{attribute 'hide_all_locals'}
FUNCTION_BLOCK DisableGroup IMPLEMENTS ITask
VAR_INPUT
END_VAR
VAR_OUTPUT
END_VAR
VAR
	groupDisable			: MC_GroupDisable;
	_caGroup			: REFERENCE TO AXES_GROUP_REF;
	State: INT;
	_disableGroup : BOOL;
	_busy : BOOL;
	_error : BOOL;
	_done : BOOL;
END_VAR

CASE State OF
	0:
		IF _disableGroup THEN
			_done := FALSE;
			_error := FALSE;
			_busy := TRUE;
			groupDisable.Execute := TRUE;
			IF groupDisable.Busy THEN
				_disableGroup := FALSE;
				State := 10;
			END_IF
		END_IF
	
	10:
		IF NOT groupDisable.Busy THEN
			IF groupDisable.Done THEN
				_done := TRUE;
			ELSIF groupDisable.Error THEN
				_error := TRUE;
			END_IF
			_busy := FALSE;
			groupDisable.Execute := false;
			State := 0;
		END_IF
END_CASE


groupDisable(AxesGroup := _caGroup);

METHOD Abort : BOOL
State := 0;
groupDisable.Execute := FALSE;
Abort := true;
END_METHOD

PROPERTY Busy : BOOL
GET
Busy := _busy;
END_GET
END_PROPERTY

PROPERTY Done : BOOL
GET
Done := _done;
END_GET
END_PROPERTY

PROPERTY Error : BOOL
GET
Error := _error;
END_GET
END_PROPERTY

METHOD Execute : BOOL
Execute := _disableGroup := TRUE;
END_METHOD

METHOD FB_init : BOOL
VAR_INPUT
	bInitRetains : BOOL; // if TRUE, the retain variables are initialized (warm start / cold start)
	bInCopyCode : BOOL;  // if TRUE, the instance afterwards gets moved into the copy code (online change)
	CAGroup : Reference TO AXES_GROUP_REF;
END_VAR
_caGroup REF= CAGroup;
END_METHOD

END_FUNCTION_BLOCK

(* stored: Version 1.1.0.1, ProductVersion 3.1.4024.6
   POU DisableGroup: Id {37828990-1151-42cb-8a82-4d653ff373ed}, SpecialFunc None
   Method Abort: Id {7caac018-1ef3-4d59-99fd-8985ed0dc129}
   Property Busy: Id {8e7df784-8a08-4f60-9919-a622643cc372}
   Get Get: Id {adafacb6-8748-4609-a08b-ba0cb1fe5dfd}
   Property Done: Id {100d7074-282d-456f-9913-da13b72dd4f2}
   Get Get: Id {d8e10206-27d6-4086-94d5-6e8e6b5bda9f}
   Property Error: Id {96349fbd-aa7b-4711-881a-35e65d26da71}
   Get Get: Id {c7cd34b3-9723-4c27-a25c-cde813d01f5c}
   Method Execute: Id {2913206c-7e61-494f-8454-3554d3c73ea6}
   Method FB_init: Id {d6523d48-61e0-479c-9063-c754da11526e} *)
